TYPE ST_FanucReq :
STRUCT
	nProgNr					:Byte;				
	nMovePoint				:BYTE;
	sName					:STRING;
END_STRUCT
END_TYPE

(* stored: Version 1.1.0.1, ProductVersion 3.1.4024.11
   DUT ST_FanucReq: Id {f1502c7e-92fb-41d5-85f8-a159c49fa577} *)
